// Mitsubishi GX Works2 project: exer  liga desliga uma entrada   PLC: Q03UDV

PROGRAM MAIN
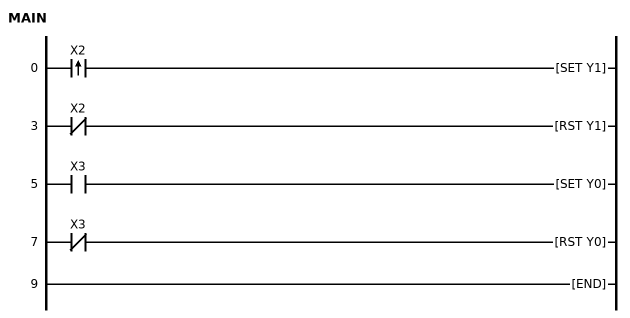
0     LDP     X2
      SET     Y1
3     LDI     X2
      RST     Y1
5     LD      X3
      SET     Y0
7     LDI     X3
      RST     Y0
9     END
END_PROGRAM
